// TIA Portal V20 export
ORGANIZATION_BLOCK "CyclicInterrupt"   // OB30, LAD, CyclicInterrupt
{ S7_Optimized_Access := 'TRUE' }
// stored: SetENOAutomatically false
   VAR_INPUT
      Initial_Call : Bool;   // Initial call of this OB
      Event_Count : Int;   // Events discarded
   END_VAR
BEGIN

REGION Network 1
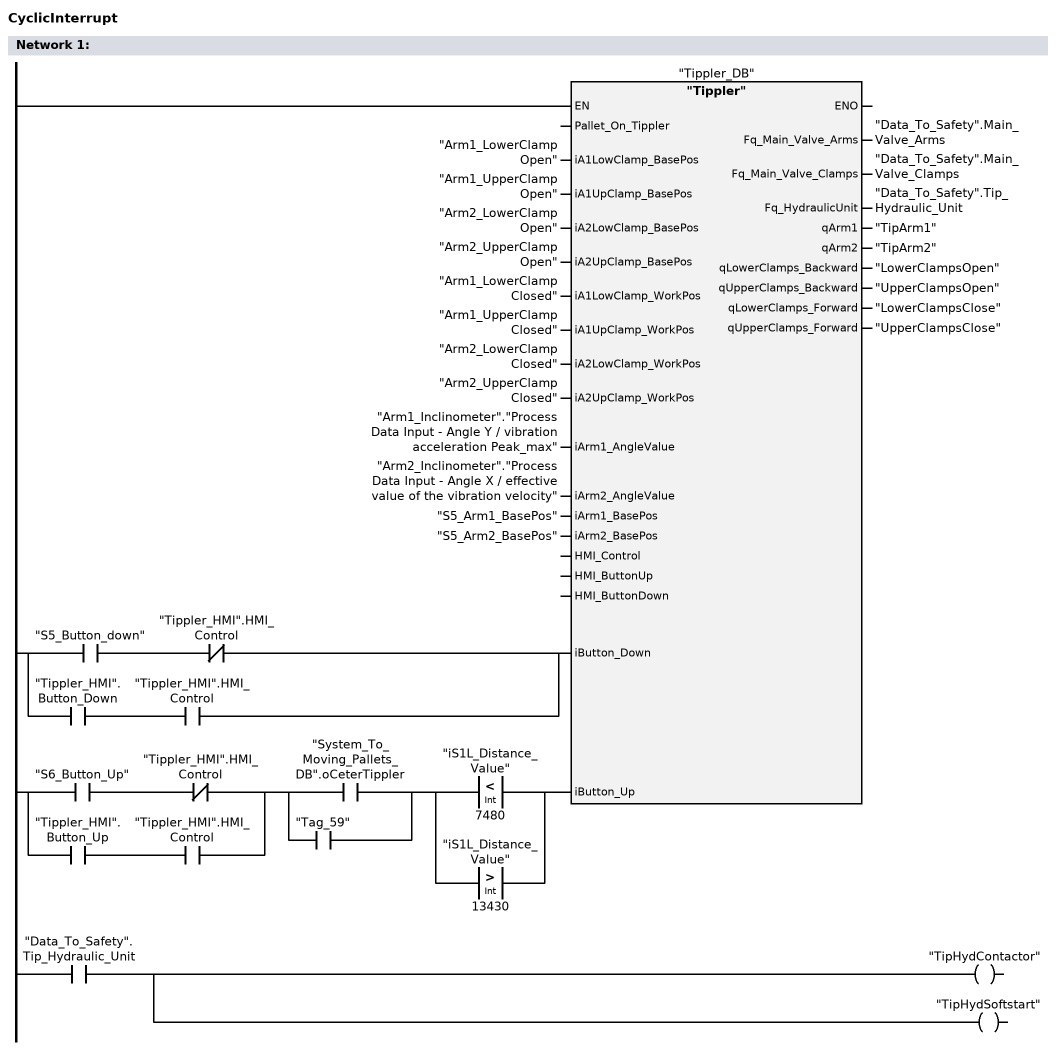
   RUNG wire#powerrail
      "Tippler_DB"(iButton_Down := wire#w1, iButton_Up := wire#w4, Pallet_On_Tippler :=, iA1LowClamp_BasePos := "Arm1_LowerClampOpen", iA1UpClamp_BasePos := "Arm1_UpperClampOpen", iA2LowClamp_BasePos := "Arm2_LowerClampOpen", iA2UpClamp_BasePos := "Arm2_UpperClampOpen", iA1LowClamp_WorkPos := "Arm1_LowerClampClosed", iA1UpClamp_WorkPos := "Arm1_UpperClampClosed", iA2LowClamp_WorkPos := "Arm2_LowerClampClosed", iA2UpClamp_WorkPos := "Arm2_UpperClampClosed", iArm1_AngleValue := "Arm1_Inclinometer"."Process Data Input - Angle Y / vibration acceleration Peak_max", iArm2_AngleValue := "Arm2_Inclinometer"."Process Data Input - Angle X / effective value of the vibration velocity", iArm1_BasePos := "S5_Arm1_BasePos", iArm2_BasePos := "S5_Arm2_BasePos", HMI_Control :=, HMI_ButtonUp :=, HMI_ButtonDown :=, Fq_Main_Valve_Arms => "Data_To_Safety".Main_Valve_Arms, Fq_Main_Valve_Clamps => "Data_To_Safety".Main_Valve_Clamps, Fq_HydraulicUnit => "Data_To_Safety".Tip_Hydraulic_Unit, qArm1 => "TipArm1", qArm2 => "TipArm2", qLowerClamps_Backward => "LowerClampsOpen", qUpperClamps_Backward => "UpperClampsOpen", qLowerClamps_Forward => "LowerClampsClose", qUpperClamps_Forward => "UpperClampsClose")
   END_RUNG
   RUNG wire#powerrail
      Contact( "S5_Button_down" )
      I_Contact( "Tippler_HMI".HMI_Control )
   END_RUNG wire#w1
   RUNG wire#powerrail
      Contact( "Tippler_HMI".Button_Down )
      Contact( "Tippler_HMI".HMI_Control )
   END_RUNG wire#w1
   RUNG wire#powerrail
      Contact( "S6_Button_Up" )
      I_Contact( "Tippler_HMI".HMI_Control )
      wire#w2
      Contact( "System_To_Moving_Pallets_DB".oCeterTippler )
      wire#w3
      { S7_Templates := "SrcType := Int" } LT_Contact(in1 := "iS1L_Distance_Value", in2 := 7480)
   END_RUNG wire#w4
   RUNG wire#powerrail
      Contact( "Tippler_HMI".Button_Up )
      Contact( "Tippler_HMI".HMI_Control )
   END_RUNG wire#w2
   RUNG wire#w2
      Contact( "Tag_59" )
   END_RUNG wire#w3
   RUNG wire#w3
      { S7_Templates := "SrcType := Int" } GT_Contact(in1 := "iS1L_Distance_Value", in2 := 13430)
   END_RUNG wire#w4
   RUNG wire#powerrail
      Contact( "Data_To_Safety".Tip_Hydraulic_Unit )
      wire#w5
      Coil( "TipHydContactor" )
   END_RUNG
   RUNG wire#w5
      Coil( "TipHydSoftstart" )
   END_RUNG
   // the same network as SCL:
   "Tippler_DB"(iA1LowClamp_BasePos := "Arm1_LowerClampOpen",   // "Tippler"
                iA1UpClamp_BasePos := "Arm1_UpperClampOpen",
                iA2LowClamp_BasePos := "Arm2_LowerClampOpen",
                iA2UpClamp_BasePos := "Arm2_UpperClampOpen",
                iA1LowClamp_WorkPos := "Arm1_LowerClampClosed",
                iA1UpClamp_WorkPos := "Arm1_UpperClampClosed",
                iA2LowClamp_WorkPos := "Arm2_LowerClampClosed",
                iA2UpClamp_WorkPos := "Arm2_UpperClampClosed",
                iArm1_AngleValue := "Arm1_Inclinometer"."Process Data Input - Angle Y / vibration acceleration Peak_max",
                iArm2_AngleValue := "Arm2_Inclinometer"."Process Data Input - Angle X / effective value of the vibration velocity",
                iArm1_BasePos := "S5_Arm1_BasePos",
                iArm2_BasePos := "S5_Arm2_BasePos",
                iButton_Down := ("S5_Button_down" AND NOT "Tippler_HMI".HMI_Control) OR ("Tippler_HMI".Button_Down AND "Tippler_HMI".HMI_Control),
                iButton_Up := (("S6_Button_Up" AND NOT "Tippler_HMI".HMI_Control) OR ("Tippler_HMI".Button_Up AND "Tippler_HMI".HMI_Control)) AND ("System_To_Moving_Pallets_DB".oCeterTippler OR "Tag_59") AND (("iS1L_Distance_Value" < 7480) OR ("iS1L_Distance_Value" > 13430)),
                Fq_Main_Valve_Arms => "Data_To_Safety".Main_Valve_Arms,
                Fq_Main_Valve_Clamps => "Data_To_Safety".Main_Valve_Clamps,
                Fq_HydraulicUnit => "Data_To_Safety".Tip_Hydraulic_Unit,
                qArm1 => "TipArm1",
                qArm2 => "TipArm2",
                qLowerClamps_Backward => "LowerClampsOpen",
                qUpperClamps_Backward => "UpperClampsOpen",
                qLowerClamps_Forward => "LowerClampsClose",
                qUpperClamps_Forward => "UpperClampsClose");
   "TipHydContactor" := "Data_To_Safety".Tip_Hydraulic_Unit;
   "TipHydSoftstart" := "Data_To_Safety".Tip_Hydraulic_Unit;
END_REGION
END_ORGANIZATION_BLOCK
